KUKA KRL program: BaseCalib.src, BaseCalib.dat

--- BaseCalib.src ---
&ACCESS RV
DEF BaseCalib ( )

END

--- BaseCalib.dat ---
&ACCESS RV
DEFDAT BaseCalib PUBLIC

ENDDAT
